(* IEC 61131-3 sources: mastertool-rankine-bridge/tests/indexer/fixtures/sample_export/objects/application_prg_0__MainPrg, 1 file *)

(* ---- declaration.st ---- *)
PROGRAM MainPrg
VAR
    xStart          : BOOL;
    xStop           : BOOL; // comentário dentro do bloco VAR
    tonAtraso       : TON;
    aiSetpoints     : ARRAY[0..3] OF INT;
END_VAR
